(* PLC project state, Beckhoff Automation GmbH TwinCAT PLC Control 3.5.13.21 *)
(* stored: creationDateTime 2024-02-04T12:47:55.1017949, modificationDateTime 2024-02-04T12:47:55.1086252 *)

{attribute 'qualified_only'}
{attribute 'strict'}
TYPE E_StateDescription :
(
	Undefined		:= 0,
	Off				:= 10,
	SelfTest		:= 20,
	Maintenance 	:= 30,
	OutOfService 	:= 40,
	Idle			:= 50,
	ServingCustomer	:= 60
);
END_TYPE

INTERFACE I_Machine
METHOD INTERNAL SetState : BOOL
VAR_INPUT
	// Set the new state to transition
	newState : I_State;
END_VAR
END_METHOD
PROPERTY IdleState : I_State
END_PROPERTY
PROPERTY MaintenanceState : I_State
END_PROPERTY
PROPERTY OffState : I_State
END_PROPERTY
PROPERTY OutOfServiceState : I_State
END_PROPERTY
PROPERTY SelfTestState : I_State
END_PROPERTY
PROPERTY ServingCustomerState : I_State
END_PROPERTY
END_INTERFACE

INTERFACE I_State
METHOD Cancel : BOOL
VAR_INPUT
END_VAR
END_METHOD
METHOD Card_Ejected : BOOL
VAR_INPUT
END_VAR
END_METHOD
METHOD Card_Inserted : BOOL
VAR_INPUT
END_VAR
END_METHOD
METHOD Failure : BOOL
VAR_INPUT
END_VAR
END_METHOD
METHOD Op : BOOL
VAR_INPUT
END_VAR
END_METHOD
METHOD Service : BOOL
VAR_INPUT
END_VAR
END_METHOD
METHOD SystemTest_OK : BOOL
VAR_INPUT
END_VAR
END_METHOD
METHOD Turn_Off : BOOL
VAR_INPUT
END_VAR
END_METHOD
METHOD Turn_On : BOOL
VAR_INPUT
END_VAR
END_METHOD
PROPERTY Description : E_StateDescription
END_PROPERTY
END_INTERFACE

FUNCTION_BLOCK FB_ATM_Machine IMPLEMENTS I_Machine
VAR_IN_OUT
	xOnButton		:	BOOL;
	xOffButton		:	BOOL;
	xServiceKey		:	BOOL;
	xCardInserted	:	BOOL;
	xCardEjected	:	BOOL;
	xCancelButton	:	BOOL;
END_VAR
VAR_OUTPUT
	ipState	:	I_State	:=	fbOff;
END_VAR
VAR
	fbOff				:	FB_Off(THIS);
	fbIdle				:	FB_Idle(THIS);
	fbMaintenance		:	FB_Maintenance(THIS);
	fbOutOfService		:	FB_OutOfService(THIS);
	fbSelfTest			:	FB_SelfTest(THIS);
	fbServingCustomer	:	FB_ServingCustomer(THIS);
	
	rtrigOnButton		:	R_TRIG;
	rtrigOffButton		:	R_TRIG;
	rtrigCancelButton	:	R_TRIG;
	rtrigCardInserted	:	R_TRIG;
	rtrigCardEjected	:	R_TRIG;
	
	// Simulation Variables
	Sim_TimerTester		:	TON 	:= (PT := T#3S);
	Sim_TimerTransaction:	TON 	:= (PT := T#3S);	
	Sim_xFaultSystem	: 	BOOL;
END_VAR

                  rtrigOnButton(CLK:= xOnButton);
rtrigOffButton(CLK:= xOffButton);
rtrigCancelButton(CLK:= xCancelButton);
rtrigCardInserted(CLK:= xCardInserted);
rtrigCardEjected(CLK:= xCardEjected);


IF rtrigOnButton.Q THEN
	ipState.Turn_On();
END_IF

IF rtrigOffButton.Q THEN
	ipState.Turn_Off();
END_IF

IF rtrigCancelButton.Q THEN
	ipState.Cancel();
END_IF

IF rtrigCardInserted.Q THEN
	ipState.Card_Inserted();
END_IF

IF rtrigCardEjected.Q THEN
	ipState.Card_Ejected();
END_IF


IF (ipState.Description = E_StateDescription.Idle OR ipState.Description = E_StateDescription.OutOfService) AND xServiceKey THEN
	ipState.Service();
END_IF

IF ipState.Description = E_StateDescription.Maintenance AND NOT xServiceKey THEN
	ipState.Op();
END_IF



// Simulation Variables - Remove and tie to I/O for moving forward
Sim_TimerTester(IN := ipState.Description = E_StateDescription.SelfTest);
IF Sim_TimerTester.Q AND NOT Sim_xFaultSystem THEN
	ipState.SystemTest_OK();
ELSIF Sim_TimerTester.Q  AND Sim_xFaultSystem THEN
	ipState.Failure();
END_IF

Sim_TimerTransaction(IN := ipState.Description = E_StateDescription.ServingCustomer);
IF Sim_TimerTransaction.Q AND NOT Sim_xFaultSystem THEN
	ipState.Card_Ejected();
ELSIF Sim_TimerTransaction.Q AND Sim_xFaultSystem THEN
	ipState.Failure();
END_IF
                

METHOD FB_Init : BOOL
VAR_INPUT
	(* if TRUE, the retain variables are initialized (warm start / cold start)*)
	bInitRetains	: BOOL;
	(* if TRUE, the instance afterwards gets moved into the copy code (online change)*)
	bInCopyCode	: BOOL;
END_VAR
                        
                      
END_METHOD

METHOD SetState : BOOL
VAR_INPUT
	(* Set the new state to transition*)
	newState	: I_State;
END_VAR
                        THIS^.ipState := newState;
                      
END_METHOD

PROPERTY IdleState : I_State
GET
VAR
END_VAR
                          IdleState := This^.fbIdle;
                        
END_GET
END_PROPERTY

PROPERTY MaintenanceState : I_State
GET
VAR
END_VAR
                          MaintenanceState := THIS^.fbMaintenance;
                        
END_GET
END_PROPERTY

PROPERTY OffState : I_State
GET
VAR
END_VAR
                          OffState := THIS^.fbOff;
                        
END_GET
END_PROPERTY

PROPERTY OutOfServiceState : I_State
GET
VAR
END_VAR
                          OutOfServiceState := THIS^.fbOutOfService;
                        
END_GET
END_PROPERTY

PROPERTY SelfTestState : I_State
GET
VAR
END_VAR
                          SelfTestState := THIS^.fbSelfTest;
                        
END_GET
END_PROPERTY

PROPERTY ServingCustomerState : I_State
GET
VAR
END_VAR
                          ServingCustomerState := THIS^.fbServingCustomer;
                        
END_GET
END_PROPERTY
END_FUNCTION_BLOCK

PROGRAM MAIN
VAR
	ATM_Machine 			: FB_ATM_Machine;
	
	xOn						:	BOOL;
	xOff					:	BOOL;
	xCancel					:	BOOL;
	xService				:	BOOL;
	xCardInserted			:	BOOL;
	xCardEjected			:	BOOL;
	ipCurrentState			:	I_State;
	CurrentStateDescription	:	STRING;


END_VAR

                  ATM_Machine(
	xOnButton:= xOn, 
	xOffButton:= xOff, 
	xCancelButton:= xCancel,
	xServiceKey	:= xService, 
	xCardInserted := xCardInserted,
	xCardEjected := xCardEjected,
	ipState=> ipCurrentState);
	
	
xOn				:= FALSE;
xOff			:= FALSE;
xCancel			:= FALSE;
xCardInserted	:= FALSE;
xCardEjected	:= FALSE;


CASE ipCurrentState.Description OF 
	E_StateDescription.Undefined :
						CurrentStateDescription := 'ATM is in undefined state, please contact the bank.';
	E_StateDescription.Off :	
						CurrentStateDescription := 'ATM is turned off.';
	E_StateDescription.SelfTest :
						CurrentStateDescription := CONCAT('ATM is in self test, current status: ', TIME_TO_STRING(ATM_Machine.Sim_TimerTester.ET));
	E_StateDescription.Maintenance : 
						CurrentStateDescription := 'Maintenance Mode';	
	E_StateDescription.OutOfService : 	
						CurrentStateDescription := 'ATM is out of service, please contact bank.';	
	E_StateDescription.Idle :			
						CurrentStateDescription := 'Please enter card or maintenance key.';	
	E_StateDescription.ServingCustomer :
						CurrentStateDescription := CONCAT('ATM is performing transaction, current status: ', TIME_TO_STRING(ATM_Machine.Sim_TimerTransaction.ET));
END_CASE                                
                
END_PROGRAM

FUNCTION_BLOCK FB_Idle IMPLEMENTS I_State
VAR_INPUT
	(* Pointer to the ATM Machine*)
	pATM_Machine	: POINTER TO FB_ATM_Machine;
END_VAR
VAR_OUTPUT
END_VAR
VAR
END_VAR

                  
                

METHOD Cancel : BOOL
                        
                      
END_METHOD

METHOD Card_Ejected : BOOL
                        
                      
END_METHOD

METHOD Card_Inserted : BOOL
                        ADSLOGSTR(ADSLOG_MSGTYPE_LOG, 'Card has been inserted!', '');
pATM_Machine^.SetState(pATM_Machine^.ServingCustomerState);
                      
END_METHOD

METHOD Failure : BOOL
                        
                      
END_METHOD

METHOD FB_Init : BOOL
VAR_INPUT
	(* if TRUE, the retain variables are initialized (warm start / cold start)*)
	bInitRetains	: BOOL;
	(* if TRUE, the instance afterwards gets moved into the copy code (online change)*)
	bInCopyCode	: BOOL;
	(* Pointer to the ATM Machine*)
	pATM_Machine	: POINTER TO FB_ATM_Machine;
END_VAR
                        THIS^.pATM_Machine := pATM_Machine;
                      
END_METHOD

METHOD Op : BOOL
                        
                      
END_METHOD

METHOD Service : BOOL
                        ADSLOGSTR(ADSLOG_MSGTYPE_LOG, 'Entering Service Mode...', '');
pATM_Machine^.SetState(pATM_Machine^.MaintenanceState);
                      
END_METHOD

METHOD SystemTest_OK : BOOL
                        
                      
END_METHOD

METHOD Turn_Off : BOOL
                        ADSLOGSTR(ADSLOG_MSGTYPE_LOG, 'Turning off machine...', '');
pATM_Machine^.SetState(pATM_Machine^.OffState);
                      
END_METHOD

METHOD Turn_On : BOOL
                        
                      
END_METHOD

PROPERTY Description : E_StateDescription
GET
VAR
END_VAR
                          Description := E_StateDescription.Idle;
                        
END_GET
END_PROPERTY
END_FUNCTION_BLOCK

FUNCTION_BLOCK FB_Maintenance IMPLEMENTS I_State
VAR_INPUT
	(* Pointer to the ATM Machine*)
	pATM_Machine	: POINTER TO FB_ATM_Machine;
END_VAR
VAR_OUTPUT
END_VAR
VAR
END_VAR

                  
                

METHOD Cancel : BOOL
                        
                      
END_METHOD

METHOD Card_Ejected : BOOL
                        
                      
END_METHOD

METHOD Card_Inserted : BOOL
                        
                      
END_METHOD

METHOD Failure : BOOL
                        
                      
END_METHOD

METHOD FB_Init : BOOL
VAR_INPUT
	(* if TRUE, the retain variables are initialized (warm start / cold start)*)
	bInitRetains	: BOOL;
	(* if TRUE, the instance afterwards gets moved into the copy code (online change)*)
	bInCopyCode	: BOOL;
	(* Pointer to the ATM Machine*)
	pATM_Machine	: POINTER TO FB_ATM_Machine;
END_VAR
                        THIS^.pATM_Machine := pATM_Machine;
                      
END_METHOD

METHOD Op : BOOL
                        ADSLOGSTR(ADSLOG_MSGTYPE_LOG, 'Exiting Service mode, going to self test', '');
pATM_Machine^.SetState(pATM_Machine^.SelfTestState);
                      
END_METHOD

METHOD Service : BOOL
                        
                      
END_METHOD

METHOD SystemTest_OK : BOOL
                        
                      
END_METHOD

METHOD Turn_Off : BOOL
                        
                      
END_METHOD

METHOD Turn_On : BOOL
                        
                      
END_METHOD

PROPERTY Description : E_StateDescription
GET
VAR
END_VAR
                          Description := E_StateDescription.Maintenance;
                        
END_GET
END_PROPERTY
END_FUNCTION_BLOCK

FUNCTION_BLOCK FB_Off IMPLEMENTS I_State
VAR_INPUT
	(* Pointer to the ATM Machine*)
	pATM_Machine	: POINTER TO FB_ATM_Machine;
END_VAR
VAR_OUTPUT
END_VAR
VAR
END_VAR

                  
                

METHOD Cancel : BOOL
                        
                      
END_METHOD

METHOD Card_Ejected : BOOL
                        
                      
END_METHOD

METHOD Card_Inserted : BOOL
                        
                      
END_METHOD

METHOD Failure : BOOL
                        
                      
END_METHOD

METHOD FB_Init : BOOL
VAR_INPUT
	(* if TRUE, the retain variables are initialized (warm start / cold start)*)
	bInitRetains	: BOOL;
	(* if TRUE, the instance afterwards gets moved into the copy code (online change)*)
	bInCopyCode	: BOOL;
	(* Pointer to the ATM Machine*)
	pATM_Machine	: POINTER TO FB_ATM_Machine;
END_VAR
                        THIS^.pATM_Machine := pATM_Machine;
                      
END_METHOD

METHOD Op : BOOL
                        
                      
END_METHOD

METHOD Service : BOOL
                        
                      
END_METHOD

METHOD SystemTest_OK : BOOL
                        
                      
END_METHOD

METHOD Turn_Off : BOOL
                        ADSLOGSTR(ADSLOG_MSGTYPE_LOG, 'Machine is already off!', '');
                      
END_METHOD

METHOD Turn_On : BOOL
                        ADSLOGSTR(ADSLOG_MSGTYPE_LOG, 'Turning on machine...', '');
pATM_Machine^.SetState(pATM_Machine^.SelfTestState);
                      
END_METHOD

PROPERTY Description : E_StateDescription
GET
VAR
END_VAR
                          Description := E_StateDescription.Off;
                        
END_GET
END_PROPERTY
END_FUNCTION_BLOCK

FUNCTION_BLOCK FB_OutOfService IMPLEMENTS I_State
VAR_INPUT
	(* Pointer to the ATM Machine*)
	pATM_Machine	: POINTER TO FB_ATM_Machine;
END_VAR
VAR_OUTPUT
END_VAR
VAR
END_VAR

                  
                

METHOD Cancel : BOOL
                        
                      
END_METHOD

METHOD Card_Ejected : BOOL
                        
                      
END_METHOD

METHOD Card_Inserted : BOOL
                        
                      
END_METHOD

METHOD Failure : BOOL
                        
                      
END_METHOD

METHOD FB_Init : BOOL
VAR_INPUT
	(* if TRUE, the retain variables are initialized (warm start / cold start)*)
	bInitRetains	: BOOL;
	(* if TRUE, the instance afterwards gets moved into the copy code (online change)*)
	bInCopyCode	: BOOL;
	(* Pointer to the ATM Machine*)
	pATM_Machine	: POINTER TO FB_ATM_Machine;
END_VAR
                        THIS^.pATM_Machine := pATM_Machine;
                      
END_METHOD

METHOD Op : BOOL
                        
                      
END_METHOD

METHOD Service : BOOL
                        ADSLOGSTR(ADSLOG_MSGTYPE_LOG, 'Entering Service Mode...', '');
pATM_Machine^.SetState(pATM_Machine^.MaintenanceState);
                      
END_METHOD

METHOD SystemTest_OK : BOOL
                        
                      
END_METHOD

METHOD Turn_Off : BOOL
                        ADSLOGSTR(ADSLOG_MSGTYPE_LOG, 'Turning off machine...', '');
pATM_Machine^.SetState(pATM_Machine^.OffState);
                      
END_METHOD

METHOD Turn_On : BOOL
                        
                      
END_METHOD

PROPERTY Description : E_StateDescription
GET
VAR
END_VAR
                          Description := E_StateDescription.OutOfService;
                        
END_GET
END_PROPERTY
END_FUNCTION_BLOCK

FUNCTION_BLOCK FB_SelfTest IMPLEMENTS I_State
VAR_INPUT
	(* Pointer to the ATM Machine*)
	pATM_Machine	: POINTER TO FB_ATM_Machine;
END_VAR
VAR_OUTPUT
END_VAR
VAR
END_VAR

                  
                

METHOD Cancel : BOOL
                        
                      
END_METHOD

METHOD Card_Ejected : BOOL
                        
                      
END_METHOD

METHOD Card_Inserted : BOOL
                        
                      
END_METHOD

METHOD Failure : BOOL
                        ADSLOGSTR(ADSLOG_MSGTYPE_LOG, 'System Test Fail, going to Out of Service', '');
pATM_Machine^.SetState(pATM_Machine^.OutOfServiceState);
                      
END_METHOD

METHOD FB_Init : BOOL
VAR_INPUT
	(* if TRUE, the retain variables are initialized (warm start / cold start)*)
	bInitRetains	: BOOL;
	(* if TRUE, the instance afterwards gets moved into the copy code (online change)*)
	bInCopyCode	: BOOL;
	(* Pointer to the ATM Machine*)
	pATM_Machine	: POINTER TO FB_ATM_Machine;
END_VAR
                        THIS^.pATM_Machine := pATM_Machine;
                      
END_METHOD

METHOD Op : BOOL
                        
                      
END_METHOD

METHOD Service : BOOL
                        
                      
END_METHOD

METHOD SystemTest_OK : BOOL
                        ADSLOGSTR(ADSLOG_MSGTYPE_LOG, 'System Test Pass, going to Idel', '');
pATM_Machine^.SetState(pATM_Machine^.IdleState);
                      
END_METHOD

METHOD Turn_Off : BOOL
                        
                      
END_METHOD

METHOD Turn_On : BOOL
                        
                      
END_METHOD

PROPERTY Description : E_StateDescription
GET
VAR
END_VAR
                          Description := E_StateDescription.SelfTest;
                        
END_GET
END_PROPERTY
END_FUNCTION_BLOCK

FUNCTION_BLOCK FB_ServingCustomer IMPLEMENTS I_State
VAR_INPUT
	(* Pointer to the ATM Machine*)
	pATM_Machine	: POINTER TO FB_ATM_Machine;
END_VAR
VAR_OUTPUT
END_VAR
VAR
END_VAR

                  
                

METHOD Cancel : BOOL
                        ADSLOGSTR(ADSLOG_MSGTYPE_LOG, 'Transaction canceled, going to idle...', '');
pATM_Machine^.SetState(pATM_Machine^.IdleState);
                      
END_METHOD

METHOD Card_Ejected : BOOL
                        ADSLOGSTR(ADSLOG_MSGTYPE_LOG, 'Card has been ejected, going to idle...', '');
pATM_Machine^.SetState(pATM_Machine^.IdleState);
                      
END_METHOD

METHOD Card_Inserted : BOOL
                        
                      
END_METHOD

METHOD Failure : BOOL
                        ADSLOGSTR(ADSLOG_MSGTYPE_LOG, 'Transaction failed, contact service...', '');
pATM_Machine^.SetState(pATM_Machine^.OutOfServiceState);
                      
END_METHOD

METHOD FB_Init : BOOL
VAR_INPUT
	(* if TRUE, the retain variables are initialized (warm start / cold start)*)
	bInitRetains	: BOOL;
	(* if TRUE, the instance afterwards gets moved into the copy code (online change)*)
	bInCopyCode	: BOOL;
	(* Pointer to the ATM Machine*)
	pATM_Machine	: POINTER TO FB_ATM_Machine;
END_VAR
                        THIS^.pATM_Machine := pATM_Machine;
                      
END_METHOD

METHOD Op : BOOL
                        
                      
END_METHOD

METHOD Service : BOOL
                        
                      
END_METHOD

METHOD SystemTest_OK : BOOL
                        
                      
END_METHOD

METHOD Turn_Off : BOOL
                        
                      
END_METHOD

METHOD Turn_On : BOOL
                        
                      
END_METHOD

PROPERTY Description : E_StateDescription
GET
VAR
END_VAR
                          Description := E_StateDescription.ServingCustomer;
                        
END_GET
END_PROPERTY
END_FUNCTION_BLOCK

CONFIGURATION Application
  RESOURCE state ON PLC
    TASK PlcTask(INTERVAL := T#0ms, PRIORITY := 20);
    PROGRAM MAIN WITH PlcTask : MAIN;
  END_RESOURCE
END_CONFIGURATION
